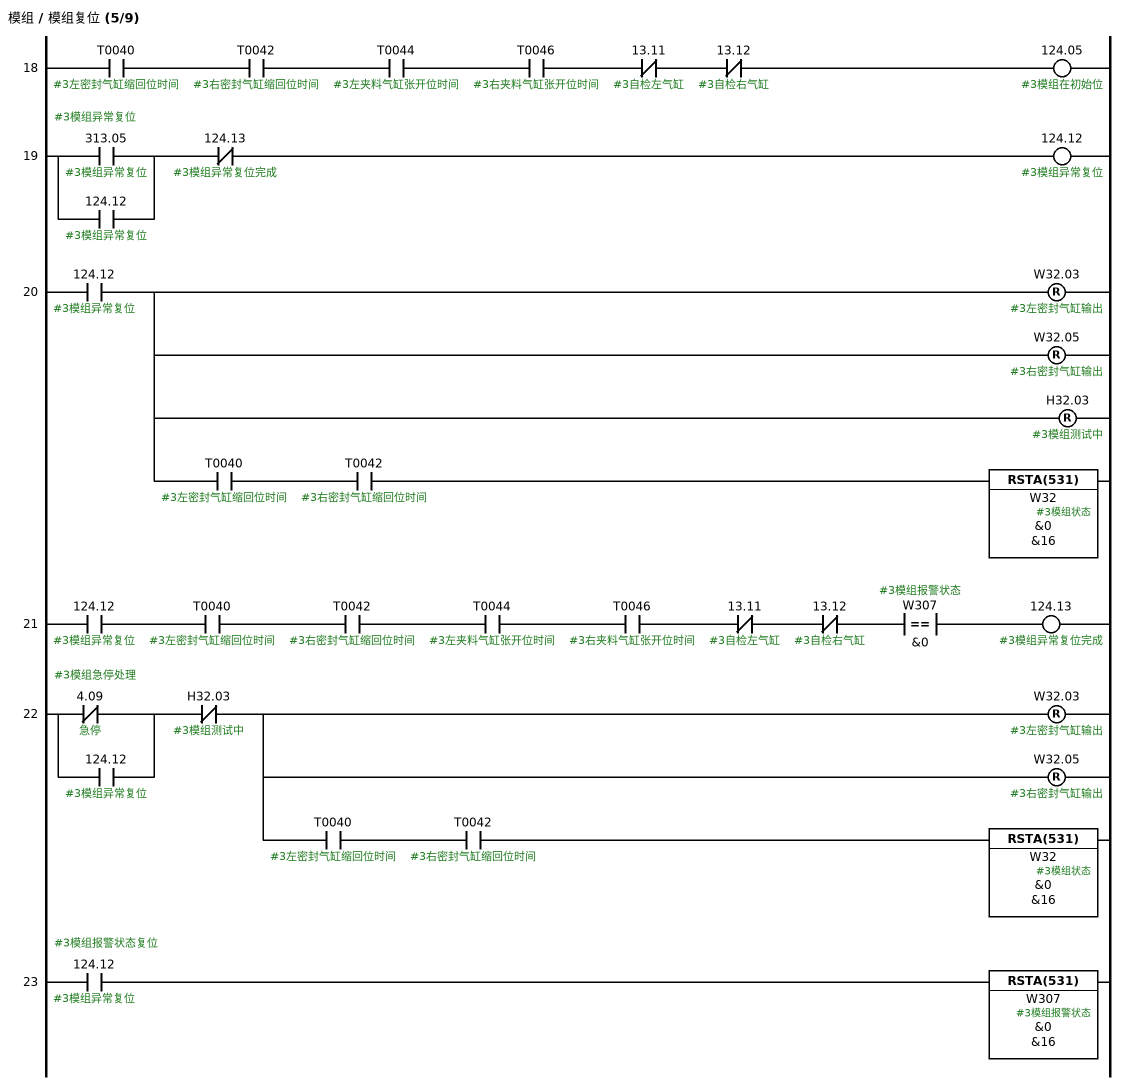
; rung 18
LD T0040  ; #3左密封气缸缩回位时间
AND T0042  ; #3右密封气缸缩回位时间
AND T0044  ; #3左夹料气缸张开位时间
AND T0046  ; #3右夹料气缸张开位时间
ANDNOT 13.11  ; #3自检左气缸
ANDNOT 13.12  ; #3自检右气缸
OUT 124.05  ; #3模组在初始位
; rung 19: #3模组异常复位
LD 313.05  ; #3模组异常复位
OR 124.12  ; #3模组异常复位
ANDNOT 124.13  ; #3模组异常复位完成
OUT 124.12  ; #3模组异常复位
; rung 20
LD 124.12  ; #3模组异常复位
RSET W32.03  ; #3左密封气缸输出
RSET W32.05  ; #3右密封气缸输出
RSET H32.03  ; #3模组测试中
AND T0040  ; #3左密封气缸缩回位时间
AND T0042  ; #3右密封气缸缩回位时间
RSTA(531) W32 &0 &16  ; #3模组状态
; rung 21
LD 124.12  ; #3模组异常复位
AND T0040  ; #3左密封气缸缩回位时间
AND T0042  ; #3右密封气缸缩回位时间
AND T0044  ; #3左夹料气缸张开位时间
AND T0046  ; #3右夹料气缸张开位时间
ANDNOT 13.11  ; #3自检左气缸
ANDNOT 13.12  ; #3自检右气缸
AND=(300) W307 &0  ; #3模组报警状态
OUT 124.13  ; #3模组异常复位完成
; rung 22: #3模组急停处理
LDNOT 4.09  ; 急停
OR 124.12  ; #3模组异常复位
ANDNOT H32.03  ; #3模组测试中
RSET W32.03  ; #3左密封气缸输出
RSET W32.05  ; #3右密封气缸输出
AND T0040  ; #3左密封气缸缩回位时间
AND T0042  ; #3右密封气缸缩回位时间
RSTA(531) W32 &0 &16  ; #3模组状态
; rung 23: #3模组报警状态复位
LD 124.12  ; #3模组异常复位
RSTA(531) W307 &0 &16  ; #3模组报警状态

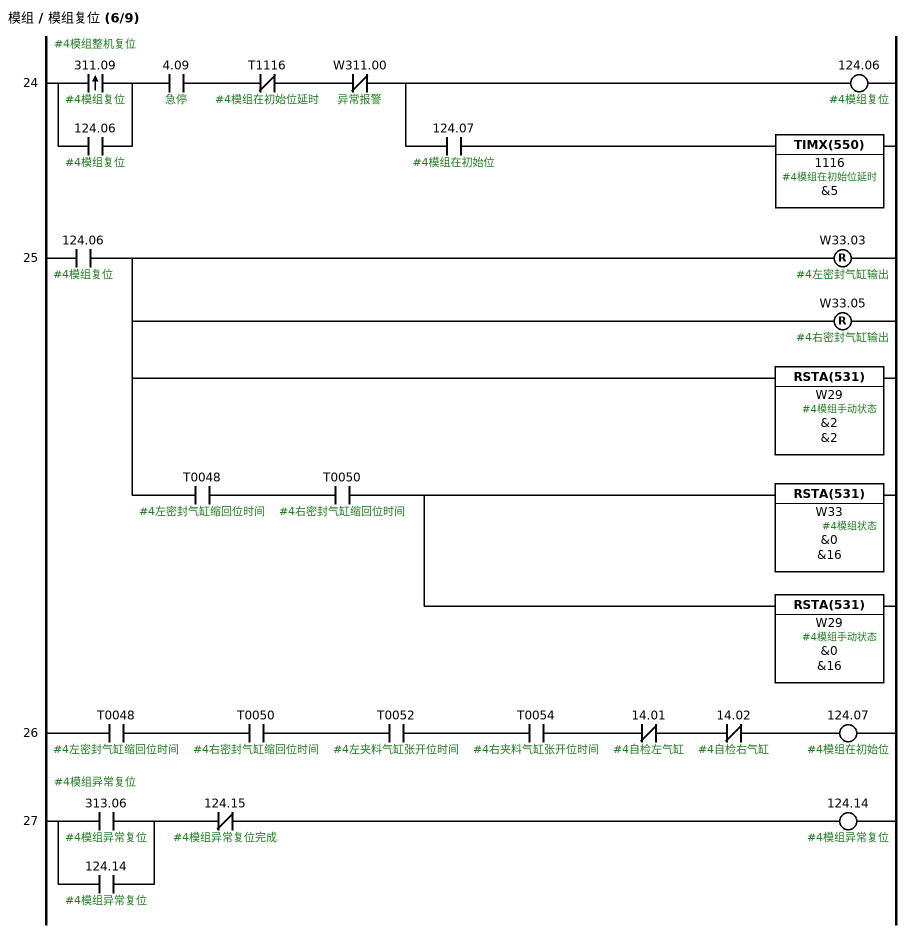
; rung 24: #4模组整机复位
@LD 311.09  ; #4模组复位
OR 124.06  ; #4模组复位
AND 4.09  ; 急停
ANDNOT T1116  ; #4模组在初始位延时
ANDNOT W311.00  ; 异常报警
OUT 124.06  ; #4模组复位
AND 124.07  ; #4模组在初始位
TIMX(550) 1116 &5  ; #4模组在初始位延时
; rung 25
LD 124.06  ; #4模组复位
RSET W33.03  ; #4左密封气缸输出
RSET W33.05  ; #4右密封气缸输出
RSTA(531) W29 &2 &2  ; #4模组手动状态
AND T0048  ; #4左密封气缸缩回位时间
AND T0050  ; #4右密封气缸缩回位时间
RSTA(531) W33 &0 &16  ; #4模组状态
RSTA(531) W29 &0 &16  ; #4模组手动状态
; rung 26
LD T0048  ; #4左密封气缸缩回位时间
AND T0050  ; #4右密封气缸缩回位时间
AND T0052  ; #4左夹料气缸张开位时间
AND T0054  ; #4右夹料气缸张开位时间
ANDNOT 14.01  ; #4自检左气缸
ANDNOT 14.02  ; #4自检右气缸
OUT 124.07  ; #4模组在初始位
; rung 27: #4模组异常复位
LD 313.06  ; #4模组异常复位
OR 124.14  ; #4模组异常复位
ANDNOT 124.15  ; #4模组异常复位完成
OUT 124.14  ; #4模组异常复位

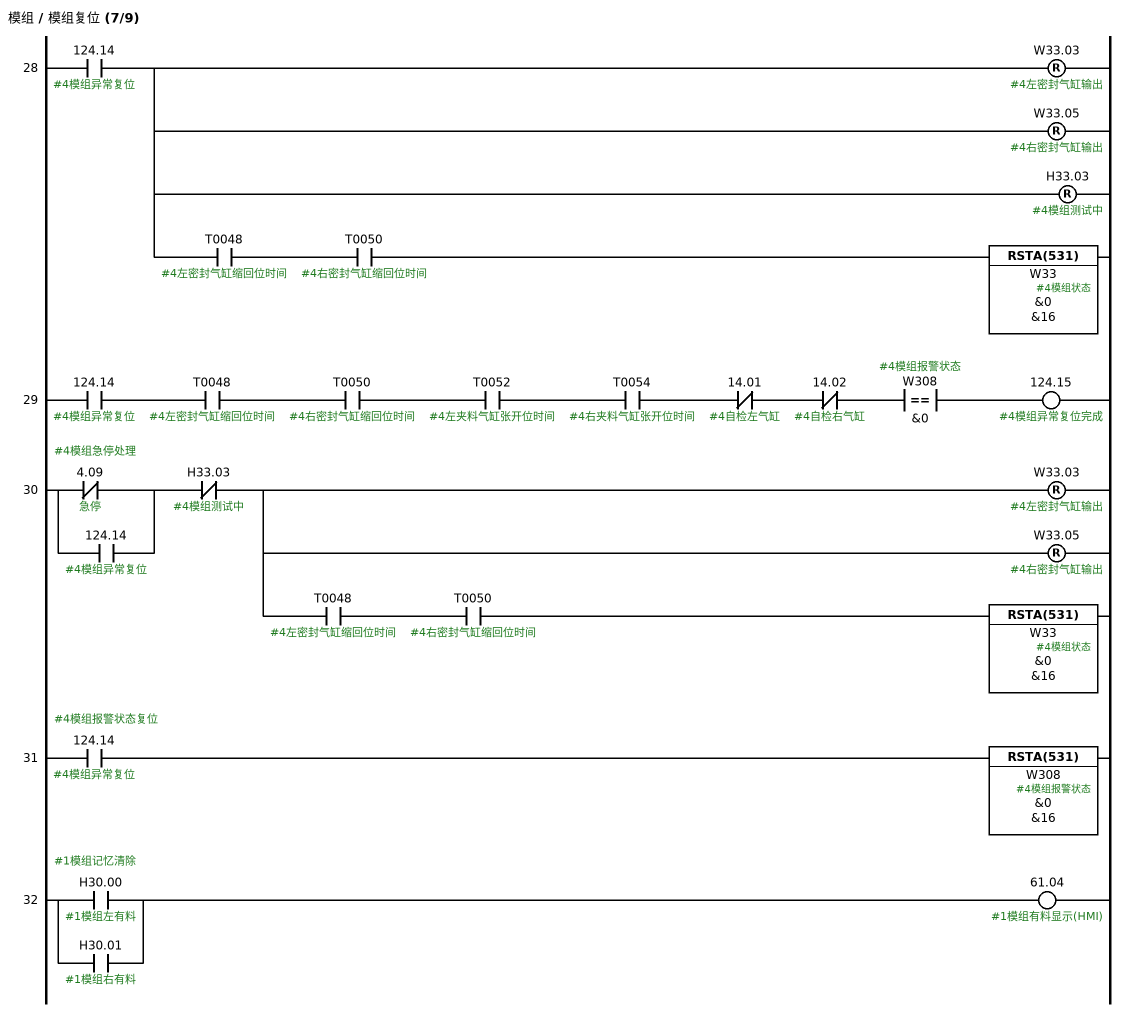
; rung 28
LD 124.14  ; #4模组异常复位
RSET W33.03  ; #4左密封气缸输出
RSET W33.05  ; #4右密封气缸输出
RSET H33.03  ; #4模组测试中
AND T0048  ; #4左密封气缸缩回位时间
AND T0050  ; #4右密封气缸缩回位时间
RSTA(531) W33 &0 &16  ; #4模组状态
; rung 29
LD 124.14  ; #4模组异常复位
AND T0048  ; #4左密封气缸缩回位时间
AND T0050  ; #4右密封气缸缩回位时间
AND T0052  ; #4左夹料气缸张开位时间
AND T0054  ; #4右夹料气缸张开位时间
ANDNOT 14.01  ; #4自检左气缸
ANDNOT 14.02  ; #4自检右气缸
AND=(300) W308 &0  ; #4模组报警状态
OUT 124.15  ; #4模组异常复位完成
; rung 30: #4模组急停处理
LDNOT 4.09  ; 急停
OR 124.14  ; #4模组异常复位
ANDNOT H33.03  ; #4模组测试中
RSET W33.03  ; #4左密封气缸输出
RSET W33.05  ; #4右密封气缸输出
AND T0048  ; #4左密封气缸缩回位时间
AND T0050  ; #4右密封气缸缩回位时间
RSTA(531) W33 &0 &16  ; #4模组状态
; rung 31: #4模组报警状态复位
LD 124.14  ; #4模组异常复位
RSTA(531) W308 &0 &16  ; #4模组报警状态
; rung 32: #1模组记忆清除
LD H30.00  ; #1模组左有料
OR H30.01  ; #1模组右有料
OUT 61.04  ; #1模组有料显示(HMI)

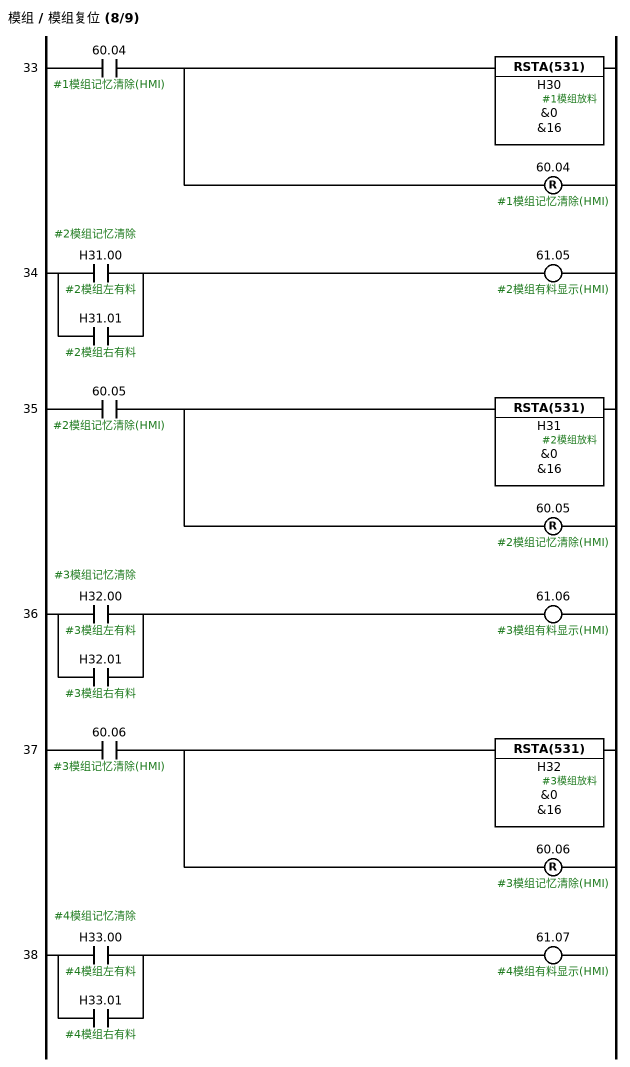
; rung 33
LD 60.04  ; #1模组记忆清除(HMI)
RSTA(531) H30 &0 &16  ; #1模组放料
RSET 60.04  ; #1模组记忆清除(HMI)
; rung 34: #2模组记忆清除
LD H31.00  ; #2模组左有料
OR H31.01  ; #2模组右有料
OUT 61.05  ; #2模组有料显示(HMI)
; rung 35
LD 60.05  ; #2模组记忆清除(HMI)
RSTA(531) H31 &0 &16  ; #2模组放料
RSET 60.05  ; #2模组记忆清除(HMI)
; rung 36: #3模组记忆清除
LD H32.00  ; #3模组左有料
OR H32.01  ; #3模组右有料
OUT 61.06  ; #3模组有料显示(HMI)
; rung 37
LD 60.06  ; #3模组记忆清除(HMI)
RSTA(531) H32 &0 &16  ; #3模组放料
RSET 60.06  ; #3模组记忆清除(HMI)
; rung 38: #4模组记忆清除
LD H33.00  ; #4模组左有料
OR H33.01  ; #4模组右有料
OUT 61.07  ; #4模组有料显示(HMI)

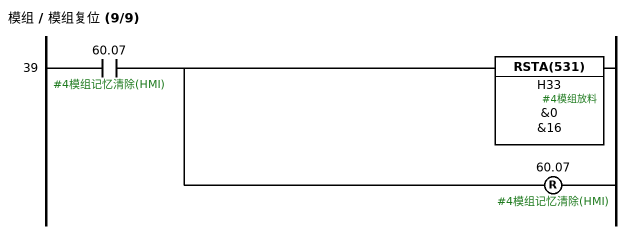
; rung 39
LD 60.07  ; #4模组记忆清除(HMI)
RSTA(531) H33 &0 &16  ; #4模组放料
RSET 60.07  ; #4模组记忆清除(HMI)

### Section END
; rung 0
END(001)

## Program 龙门机械手 (cyclic task 7)
Local symbols
P_on BOOL

### Section 龙门、料盒升降手动

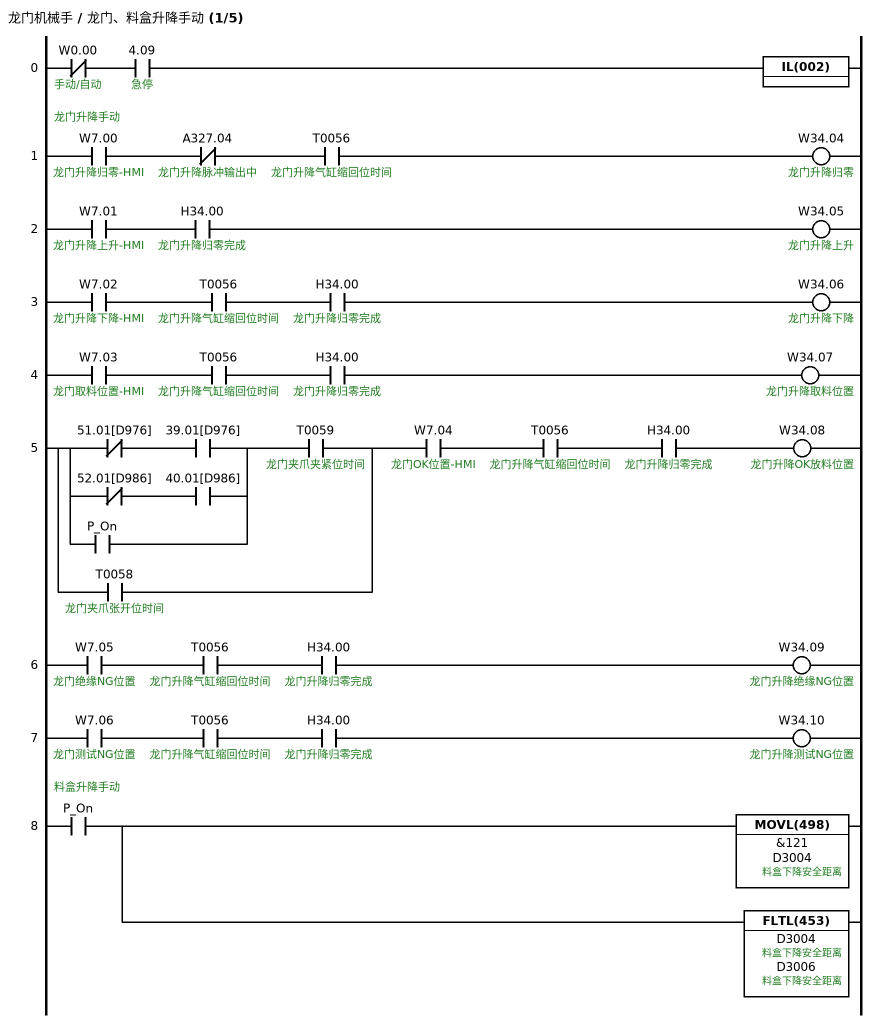
; rung 0
LDNOT W0.00  ; 手动/自动
AND 4.09  ; 急停
IL(002)
; rung 1: 龙门升降手动
LD W7.00  ; 龙门升降归零-HMI
ANDNOT A327.04  ; 龙门升降脉冲输出中
AND T0056  ; 龙门升降气缸缩回位时间
OUT W34.04  ; 龙门升降归零
; rung 2
LD W7.01  ; 龙门升降上升-HMI
AND H34.00  ; 龙门升降归零完成
OUT W34.05  ; 龙门升降上升
; rung 3
LD W7.02  ; 龙门升降下降-HMI
AND T0056  ; 龙门升降气缸缩回位时间
AND H34.00  ; 龙门升降归零完成
OUT W34.06  ; 龙门升降下降
; rung 4
LD W7.03  ; 龙门取料位置-HMI
AND T0056  ; 龙门升降气缸缩回位时间
AND H34.00  ; 龙门升降归零完成
OUT W34.07  ; 龙门升降取料位置
; rung 5
LDNOT 51.01[D976]
AND 39.01[D976]
LDNOT 52.01[D986]
AND 40.01[D986]
ORLD
OR P_On
AND T0059  ; 龙门夹爪夹紧位时间
OR T0058  ; 龙门夹爪张开位时间
AND W7.04  ; 龙门OK位置-HMI
AND T0056  ; 龙门升降气缸缩回位时间
AND H34.00  ; 龙门升降归零完成
OUT W34.08  ; 龙门升降OK放料位置
; rung 6
LD W7.05  ; 龙门绝缘NG位置
AND T0056  ; 龙门升降气缸缩回位时间
AND H34.00  ; 龙门升降归零完成
OUT W34.09  ; 龙门升降绝缘NG位置
; rung 7
LD W7.06  ; 龙门测试NG位置
AND T0056  ; 龙门升降气缸缩回位时间
AND H34.00  ; 龙门升降归零完成
OUT W34.10  ; 龙门升降测试NG位置
; rung 8: 料盒升降手动
LD P_On
MOVL(498) &121 D3004  ; 料盒下降安全距离
FLTL(453) D3004 D3006  ; 料盒下降安全距离

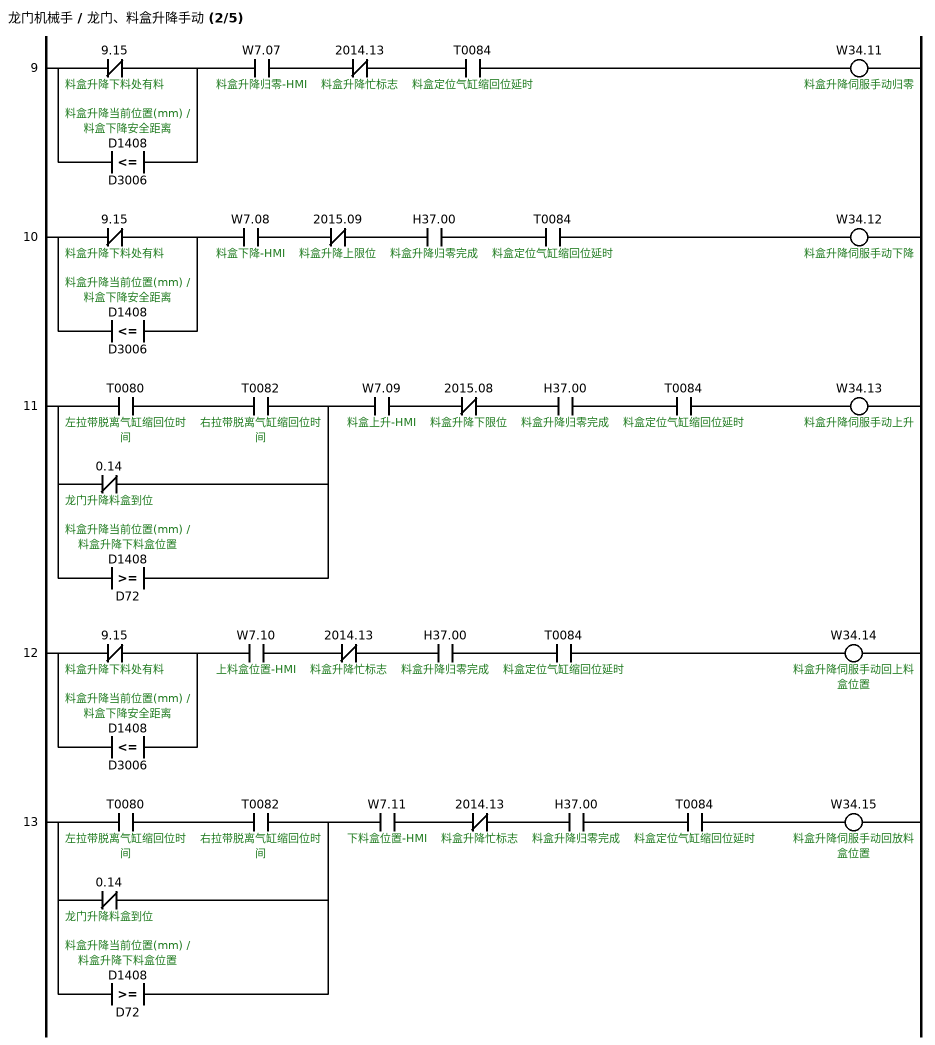
; rung 9
LDNOT 9.15  ; 料盒升降下料处有料
OR<=F(332) D1408 D3006  ; 料盒升降当前位置(mm), 料盒下降安全距离
AND W7.07  ; 料盒升降归零-HMI
ANDNOT 2014.13  ; 料盒升降忙标志
AND T0084  ; 料盒定位气缸缩回位延时
OUT W34.11  ; 料盒升降伺服手动归零
; rung 10
LDNOT 9.15  ; 料盒升降下料处有料
OR<=F(332) D1408 D3006  ; 料盒升降当前位置(mm), 料盒下降安全距离
AND W7.08  ; 料盒下降-HMI
ANDNOT 2015.09  ; 料盒升降上限位
AND H37.00  ; 料盒升降归零完成
AND T0084  ; 料盒定位气缸缩回位延时
OUT W34.12  ; 料盒升降伺服手动下降
; rung 11
LD T0080  ; 左拉带脱离气缸缩回位时间
AND T0082  ; 右拉带脱离气缸缩回位时间
ORNOT 0.14  ; 龙门升降料盒到位
OR>=F(334) D1408 D72  ; 料盒升降当前位置(mm), 料盒升降下料盒位置
AND W7.09  ; 料盒上升-HMI
ANDNOT 2015.08  ; 料盒升降下限位
AND H37.00  ; 料盒升降归零完成
AND T0084  ; 料盒定位气缸缩回位延时
OUT W34.13  ; 料盒升降伺服手动上升
; rung 12
LDNOT 9.15  ; 料盒升降下料处有料
OR<=F(332) D1408 D3006  ; 料盒升降当前位置(mm), 料盒下降安全距离
AND W7.10  ; 上料盒位置-HMI
ANDNOT 2014.13  ; 料盒升降忙标志
AND H37.00  ; 料盒升降归零完成
AND T0084  ; 料盒定位气缸缩回位延时
OUT W34.14  ; 料盒升降伺服手动回上料盒位置
; rung 13
LD T0080  ; 左拉带脱离气缸缩回位时间
AND T0082  ; 右拉带脱离气缸缩回位时间
ORNOT 0.14  ; 龙门升降料盒到位
OR>=F(334) D1408 D72  ; 料盒升降当前位置(mm), 料盒升降下料盒位置
AND W7.11  ; 下料盒位置-HMI
ANDNOT 2014.13  ; 料盒升降忙标志
AND H37.00  ; 料盒升降归零完成
AND T0084  ; 料盒定位气缸缩回位延时
OUT W34.15  ; 料盒升降伺服手动回放料盒位置

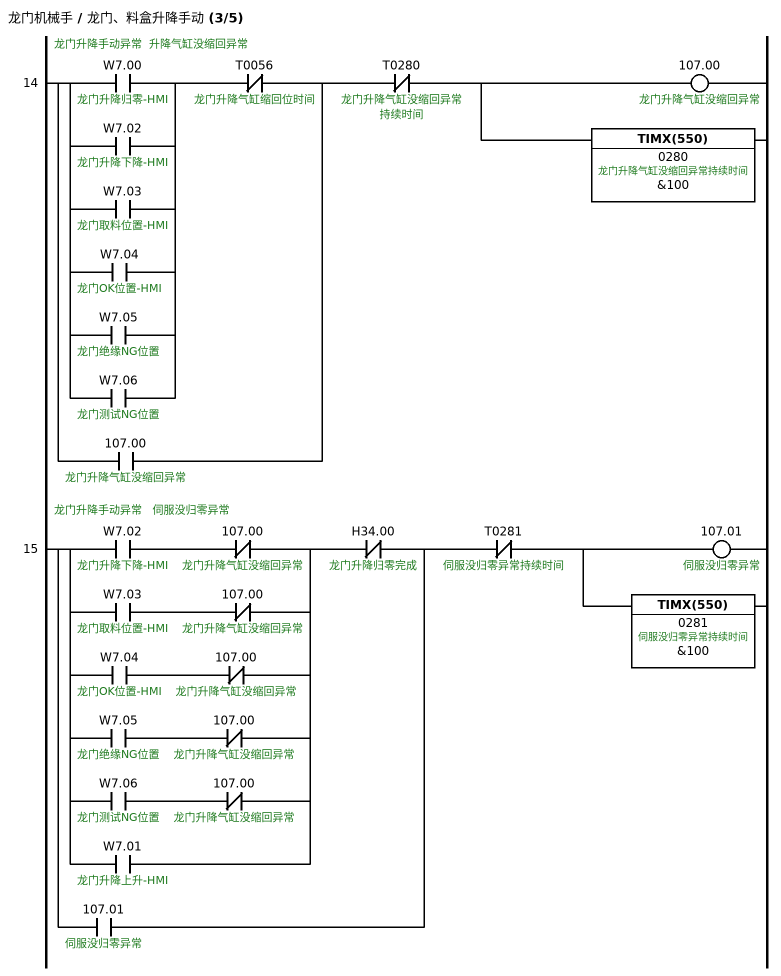
; rung 14: 龙门升降手动异常  升降气缸没缩回异常
LD W7.00  ; 龙门升降归零-HMI
OR W7.02  ; 龙门升降下降-HMI
OR W7.03  ; 龙门取料位置-HMI
OR W7.04  ; 龙门OK位置-HMI
OR W7.05  ; 龙门绝缘NG位置
OR W7.06  ; 龙门测试NG位置
ANDNOT T0056  ; 龙门升降气缸缩回位时间
OR 107.00  ; 龙门升降气缸没缩回异常
ANDNOT T0280  ; 龙门升降气缸没缩回异常持续时间
OUT 107.00  ; 龙门升降气缸没缩回异常
TIMX(550) 0280 &100  ; 龙门升降气缸没缩回异常持续时间
; rung 15: 龙门升降手动异常   伺服没归零异常
LD W7.02  ; 龙门升降下降-HMI
ANDNOT 107.00  ; 龙门升降气缸没缩回异常
LD W7.03  ; 龙门取料位置-HMI
ANDNOT 107.00  ; 龙门升降气缸没缩回异常
ORLD
LD W7.04  ; 龙门OK位置-HMI
ANDNOT 107.00  ; 龙门升降气缸没缩回异常
ORLD
LD W7.05  ; 龙门绝缘NG位置
ANDNOT 107.00  ; 龙门升降气缸没缩回异常
ORLD
LD W7.06  ; 龙门测试NG位置
ANDNOT 107.00  ; 龙门升降气缸没缩回异常
ORLD
OR W7.01  ; 龙门升降上升-HMI
ANDNOT H34.00  ; 龙门升降归零完成
OR 107.01  ; 伺服没归零异常
ANDNOT T0281  ; 伺服没归零异常持续时间
OUT 107.01  ; 伺服没归零异常
TIMX(550) 0281 &100  ; 伺服没归零异常持续时间

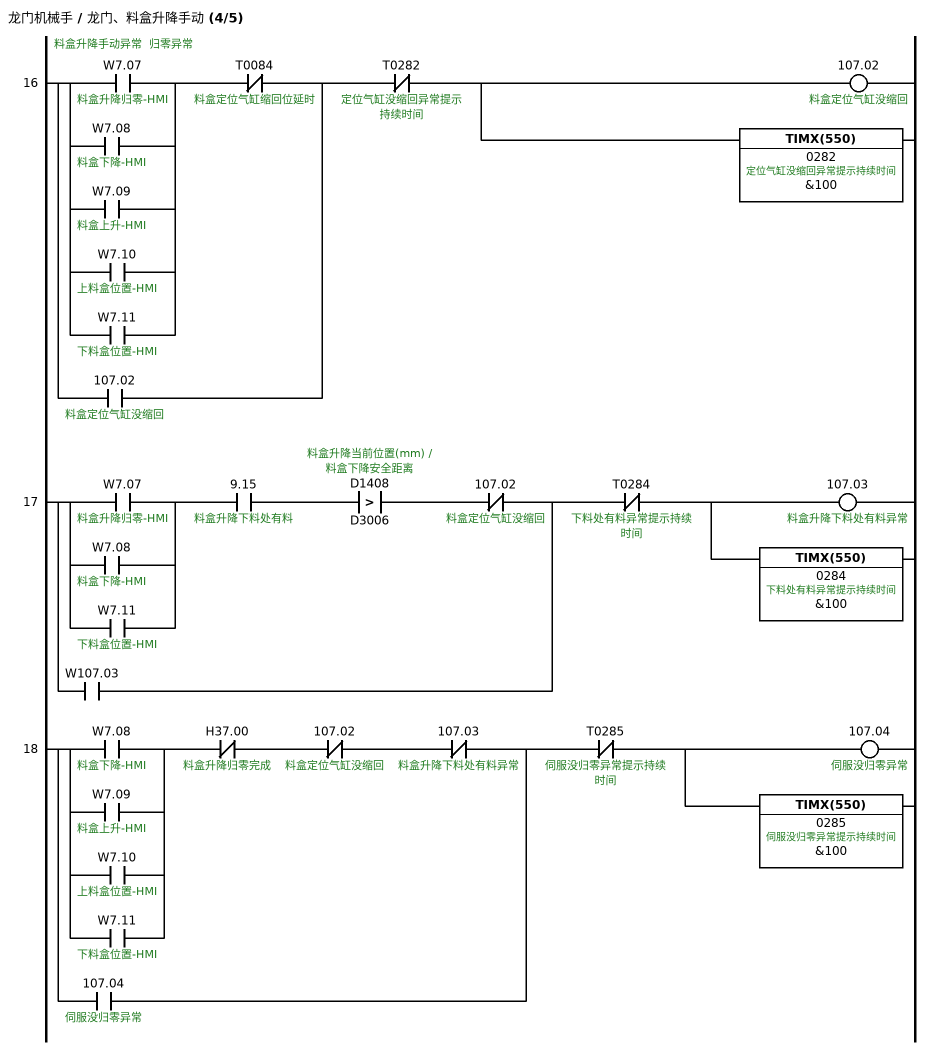
; rung 16: 料盒升降手动异常  归零异常
LD W7.07  ; 料盒升降归零-HMI
OR W7.08  ; 料盒下降-HMI
OR W7.09  ; 料盒上升-HMI
OR W7.10  ; 上料盒位置-HMI
OR W7.11  ; 下料盒位置-HMI
ANDNOT T0084  ; 料盒定位气缸缩回位延时
OR 107.02  ; 料盒定位气缸没缩回
ANDNOT T0282  ; 定位气缸没缩回异常提示持续时间
OUT 107.02  ; 料盒定位气缸没缩回
TIMX(550) 0282 &100  ; 定位气缸没缩回异常提示持续时间
; rung 17
LD W7.07  ; 料盒升降归零-HMI
OR W7.08  ; 料盒下降-HMI
OR W7.11  ; 下料盒位置-HMI
AND 9.15  ; 料盒升降下料处有料
AND>F(333) D1408 D3006  ; 料盒升降当前位置(mm), 料盒下降安全距离
ANDNOT 107.02  ; 料盒定位气缸没缩回
OR W107.03
ANDNOT T0284  ; 下料处有料异常提示持续时间
OUT 107.03  ; 料盒升降下料处有料异常
TIMX(550) 0284 &100  ; 下料处有料异常提示持续时间
; rung 18
LD W7.08  ; 料盒下降-HMI
OR W7.09  ; 料盒上升-HMI
OR W7.10  ; 上料盒位置-HMI
OR W7.11  ; 下料盒位置-HMI
ANDNOT H37.00  ; 料盒升降归零完成
ANDNOT 107.02  ; 料盒定位气缸没缩回
ANDNOT 107.03  ; 料盒升降下料处有料异常
OR 107.04  ; 伺服没归零异常
ANDNOT T0285  ; 伺服没归零异常提示持续时间
OUT 107.04  ; 伺服没归零异常
TIMX(550) 0285 &100  ; 伺服没归零异常提示持续时间

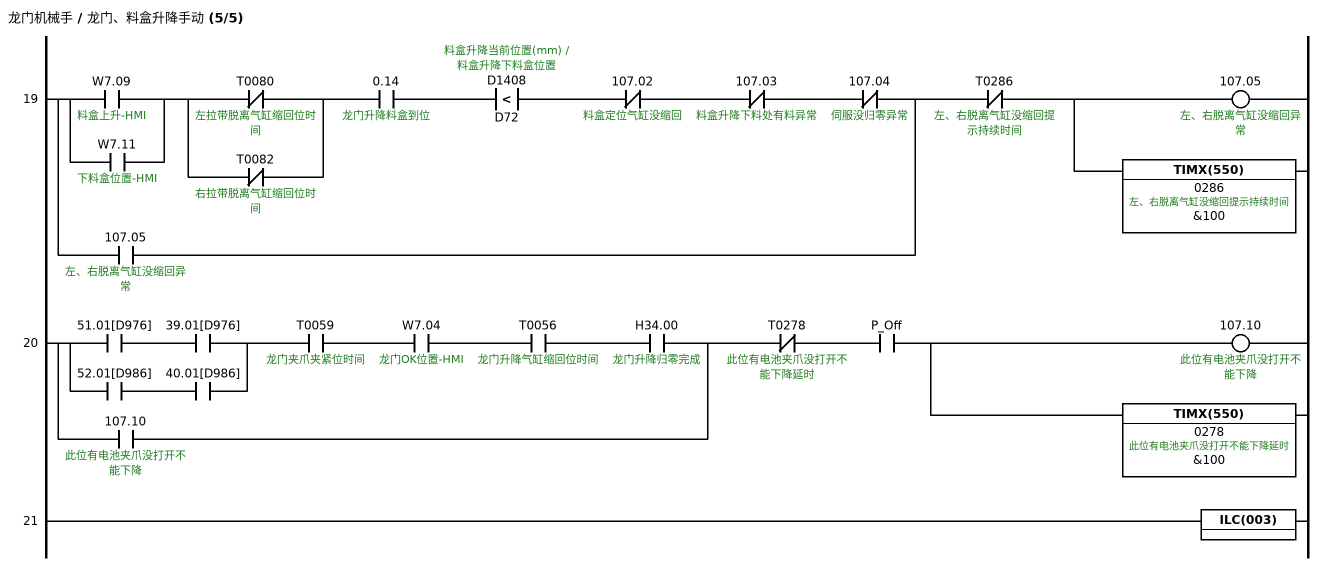
; rung 19
LD W7.09  ; 料盒上升-HMI
OR W7.11  ; 下料盒位置-HMI
LDNOT T0080  ; 左拉带脱离气缸缩回位时间
ORNOT T0082  ; 右拉带脱离气缸缩回位时间
ANDLD
AND 0.14  ; 龙门升降料盒到位
AND<F(331) D1408 D72  ; 料盒升降当前位置(mm), 料盒升降下料盒位置
ANDNOT 107.02  ; 料盒定位气缸没缩回
ANDNOT 107.03  ; 料盒升降下料处有料异常
ANDNOT 107.04  ; 伺服没归零异常
OR 107.05  ; 左、右脱离气缸没缩回异常
ANDNOT T0286  ; 左、右脱离气缸没缩回提示持续时间
OUT 107.05  ; 左、右脱离气缸没缩回异常
TIMX(550) 0286 &100  ; 左、右脱离气缸没缩回提示持续时间
; rung 20
LD 51.01[D976]
AND 39.01[D976]
LD 52.01[D986]
AND 40.01[D986]
ORLD
AND T0059  ; 龙门夹爪夹紧位时间
AND W7.04  ; 龙门OK位置-HMI
AND T0056  ; 龙门升降气缸缩回位时间
AND H34.00  ; 龙门升降归零完成
OR 107.10  ; 此位有电池夹爪没打开不能下降
ANDNOT T0278  ; 此位有电池夹爪没打开不能下降延时
AND P_Off
OUT 107.10  ; 此位有电池夹爪没打开不能下降
TIMX(550) 0278 &100  ; 此位有电池夹爪没打开不能下降延时
; rung 21
ILC(003)

### Section 龙门前后、左右手动

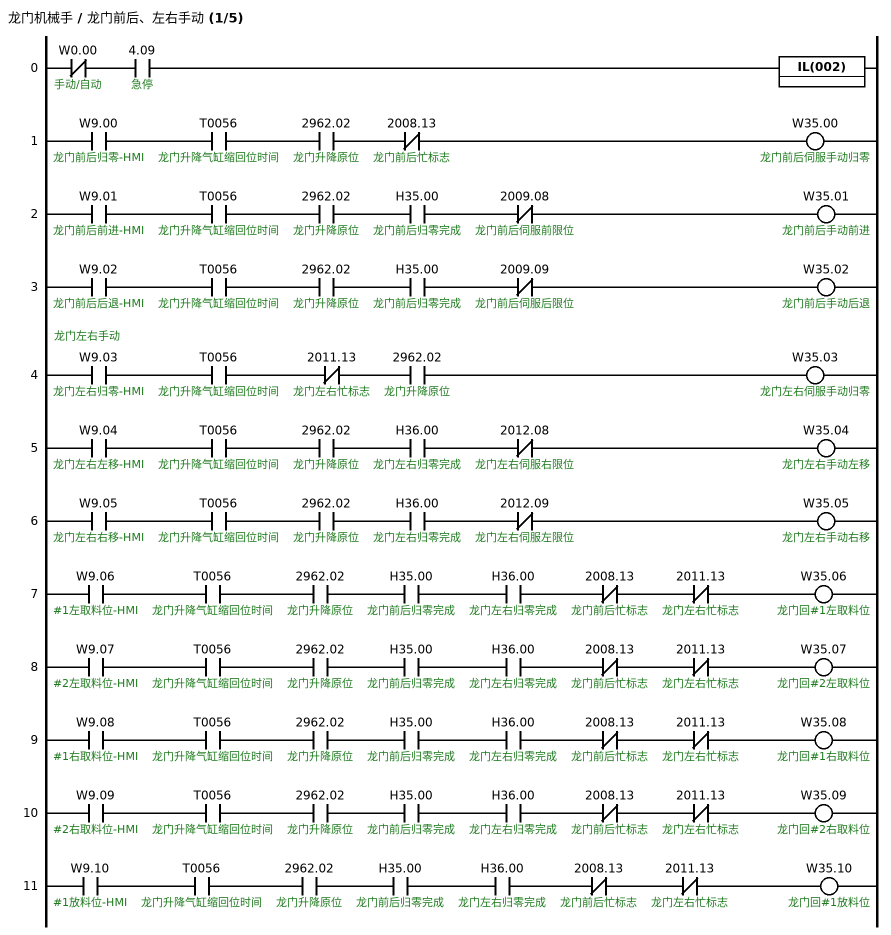
; rung 0
LDNOT W0.00  ; 手动/自动
AND 4.09  ; 急停
IL(002)
; rung 1
LD W9.00  ; 龙门前后归零-HMI
AND T0056  ; 龙门升降气缸缩回位时间
AND 2962.02  ; 龙门升降原位
ANDNOT 2008.13  ; 龙门前后忙标志
OUT W35.00  ; 龙门前后伺服手动归零
; rung 2
LD W9.01  ; 龙门前后前进-HMI
AND T0056  ; 龙门升降气缸缩回位时间
AND 2962.02  ; 龙门升降原位
AND H35.00  ; 龙门前后归零完成
ANDNOT 2009.08  ; 龙门前后伺服前限位
OUT W35.01  ; 龙门前后手动前进
; rung 3
LD W9.02  ; 龙门前后后退-HMI
AND T0056  ; 龙门升降气缸缩回位时间
AND 2962.02  ; 龙门升降原位
AND H35.00  ; 龙门前后归零完成
ANDNOT 2009.09  ; 龙门前后伺服后限位
OUT W35.02  ; 龙门前后手动后退
; rung 4: 龙门左右手动
LD W9.03  ; 龙门左右归零-HMI
AND T0056  ; 龙门升降气缸缩回位时间
ANDNOT 2011.13  ; 龙门左右忙标志
AND 2962.02  ; 龙门升降原位
OUT W35.03  ; 龙门左右伺服手动归零
; rung 5
LD W9.04  ; 龙门左右左移-HMI
AND T0056  ; 龙门升降气缸缩回位时间
AND 2962.02  ; 龙门升降原位
AND H36.00  ; 龙门左右归零完成
ANDNOT 2012.08  ; 龙门左右伺服右限位
OUT W35.04  ; 龙门左右手动左移
; rung 6
LD W9.05  ; 龙门左右右移-HMI
AND T0056  ; 龙门升降气缸缩回位时间
AND 2962.02  ; 龙门升降原位
AND H36.00  ; 龙门左右归零完成
ANDNOT 2012.09  ; 龙门左右伺服左限位
OUT W35.05  ; 龙门左右手动右移
; rung 7
LD W9.06  ; #1左取料位-HMI
AND T0056  ; 龙门升降气缸缩回位时间
AND 2962.02  ; 龙门升降原位
AND H35.00  ; 龙门前后归零完成
AND H36.00  ; 龙门左右归零完成
ANDNOT 2008.13  ; 龙门前后忙标志
ANDNOT 2011.13  ; 龙门左右忙标志
OUT W35.06  ; 龙门回#1左取料位
; rung 8
LD W9.07  ; #2左取料位-HMI
AND T0056  ; 龙门升降气缸缩回位时间
AND 2962.02  ; 龙门升降原位
AND H35.00  ; 龙门前后归零完成
AND H36.00  ; 龙门左右归零完成
ANDNOT 2008.13  ; 龙门前后忙标志
ANDNOT 2011.13  ; 龙门左右忙标志
OUT W35.07  ; 龙门回#2左取料位
; rung 9
LD W9.08  ; #1右取料位-HMI
AND T0056  ; 龙门升降气缸缩回位时间
AND 2962.02  ; 龙门升降原位
AND H35.00  ; 龙门前后归零完成
AND H36.00  ; 龙门左右归零完成
ANDNOT 2008.13  ; 龙门前后忙标志
ANDNOT 2011.13  ; 龙门左右忙标志
OUT W35.08  ; 龙门回#1右取料位
; rung 10
LD W9.09  ; #2右取料位-HMI
AND T0056  ; 龙门升降气缸缩回位时间
AND 2962.02  ; 龙门升降原位
AND H35.00  ; 龙门前后归零完成
AND H36.00  ; 龙门左右归零完成
ANDNOT 2008.13  ; 龙门前后忙标志
ANDNOT 2011.13  ; 龙门左右忙标志
OUT W35.09  ; 龙门回#2右取料位
; rung 11
LD W9.10  ; #1放料位-HMI
AND T0056  ; 龙门升降气缸缩回位时间
AND 2962.02  ; 龙门升降原位
AND H35.00  ; 龙门前后归零完成
AND H36.00  ; 龙门左右归零完成
ANDNOT 2008.13  ; 龙门前后忙标志
ANDNOT 2011.13  ; 龙门左右忙标志
OUT W35.10  ; 龙门回#1放料位

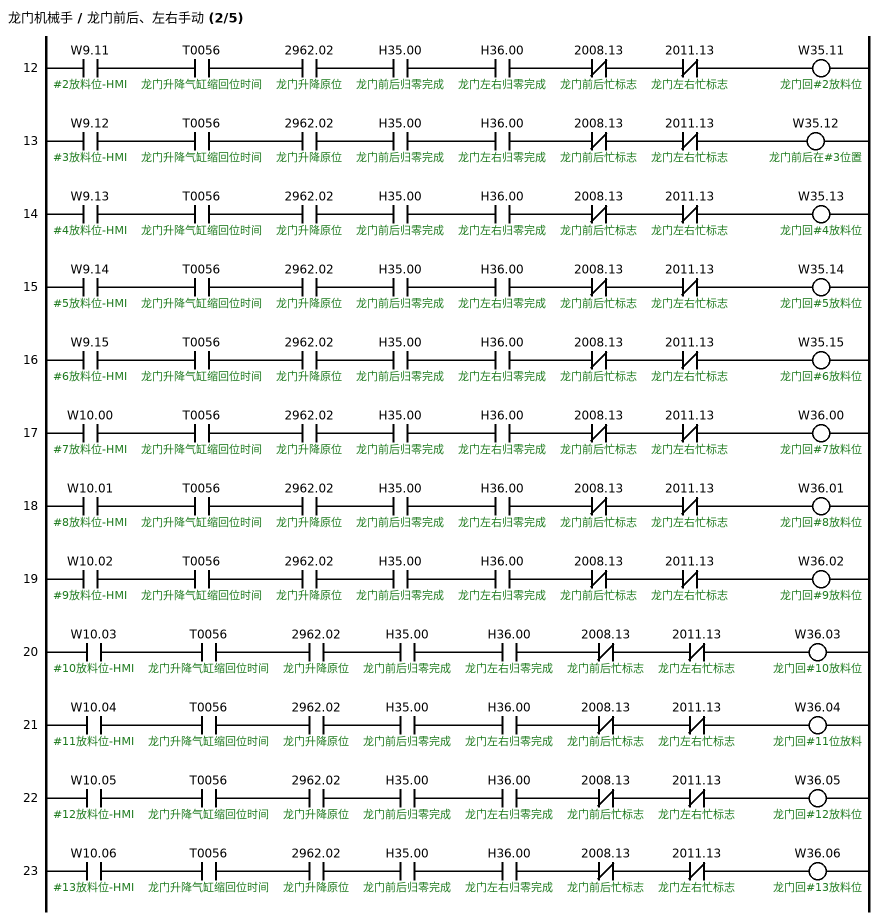
; rung 12
LD W9.11  ; #2放料位-HMI
AND T0056  ; 龙门升降气缸缩回位时间
AND 2962.02  ; 龙门升降原位
AND H35.00  ; 龙门前后归零完成
AND H36.00  ; 龙门左右归零完成
ANDNOT 2008.13  ; 龙门前后忙标志
ANDNOT 2011.13  ; 龙门左右忙标志
OUT W35.11  ; 龙门回#2放料位
; rung 13
LD W9.12  ; #3放料位-HMI
AND T0056  ; 龙门升降气缸缩回位时间
AND 2962.02  ; 龙门升降原位
AND H35.00  ; 龙门前后归零完成
AND H36.00  ; 龙门左右归零完成
ANDNOT 2008.13  ; 龙门前后忙标志
ANDNOT 2011.13  ; 龙门左右忙标志
OUT W35.12  ; 龙门前后在#3位置
; rung 14
LD W9.13  ; #4放料位-HMI
AND T0056  ; 龙门升降气缸缩回位时间
AND 2962.02  ; 龙门升降原位
AND H35.00  ; 龙门前后归零完成
AND H36.00  ; 龙门左右归零完成
ANDNOT 2008.13  ; 龙门前后忙标志
ANDNOT 2011.13  ; 龙门左右忙标志
OUT W35.13  ; 龙门回#4放料位
; rung 15
LD W9.14  ; #5放料位-HMI
AND T0056  ; 龙门升降气缸缩回位时间
AND 2962.02  ; 龙门升降原位
AND H35.00  ; 龙门前后归零完成
AND H36.00  ; 龙门左右归零完成
ANDNOT 2008.13  ; 龙门前后忙标志
ANDNOT 2011.13  ; 龙门左右忙标志
OUT W35.14  ; 龙门回#5放料位
; rung 16
LD W9.15  ; #6放料位-HMI
AND T0056  ; 龙门升降气缸缩回位时间
AND 2962.02  ; 龙门升降原位
AND H35.00  ; 龙门前后归零完成
AND H36.00  ; 龙门左右归零完成
ANDNOT 2008.13  ; 龙门前后忙标志
ANDNOT 2011.13  ; 龙门左右忙标志
OUT W35.15  ; 龙门回#6放料位
; rung 17
LD W10.00  ; #7放料位-HMI
AND T0056  ; 龙门升降气缸缩回位时间
AND 2962.02  ; 龙门升降原位
AND H35.00  ; 龙门前后归零完成
AND H36.00  ; 龙门左右归零完成
ANDNOT 2008.13  ; 龙门前后忙标志
ANDNOT 2011.13  ; 龙门左右忙标志
OUT W36.00  ; 龙门回#7放料位
; rung 18
LD W10.01  ; #8放料位-HMI
AND T0056  ; 龙门升降气缸缩回位时间
AND 2962.02  ; 龙门升降原位
AND H35.00  ; 龙门前后归零完成
AND H36.00  ; 龙门左右归零完成
ANDNOT 2008.13  ; 龙门前后忙标志
ANDNOT 2011.13  ; 龙门左右忙标志
OUT W36.01  ; 龙门回#8放料位
; rung 19
LD W10.02  ; #9放料位-HMI
AND T0056  ; 龙门升降气缸缩回位时间
AND 2962.02  ; 龙门升降原位
AND H35.00  ; 龙门前后归零完成
AND H36.00  ; 龙门左右归零完成
ANDNOT 2008.13  ; 龙门前后忙标志
ANDNOT 2011.13  ; 龙门左右忙标志
OUT W36.02  ; 龙门回#9放料位
; rung 20
LD W10.03  ; #10放料位-HMI
AND T0056  ; 龙门升降气缸缩回位时间
AND 2962.02  ; 龙门升降原位
AND H35.00  ; 龙门前后归零完成
AND H36.00  ; 龙门左右归零完成
ANDNOT 2008.13  ; 龙门前后忙标志
ANDNOT 2011.13  ; 龙门左右忙标志
OUT W36.03  ; 龙门回#10放料位
; rung 21
LD W10.04  ; #11放料位-HMI
AND T0056  ; 龙门升降气缸缩回位时间
AND 2962.02  ; 龙门升降原位
AND H35.00  ; 龙门前后归零完成
AND H36.00  ; 龙门左右归零完成
ANDNOT 2008.13  ; 龙门前后忙标志
ANDNOT 2011.13  ; 龙门左右忙标志
OUT W36.04  ; 龙门回#11位放料
; rung 22
LD W10.05  ; #12放料位-HMI
AND T0056  ; 龙门升降气缸缩回位时间
AND 2962.02  ; 龙门升降原位
AND H35.00  ; 龙门前后归零完成
AND H36.00  ; 龙门左右归零完成
ANDNOT 2008.13  ; 龙门前后忙标志
ANDNOT 2011.13  ; 龙门左右忙标志
OUT W36.05  ; 龙门回#12放料位
; rung 23
LD W10.06  ; #13放料位-HMI
AND T0056  ; 龙门升降气缸缩回位时间
AND 2962.02  ; 龙门升降原位
AND H35.00  ; 龙门前后归零完成
AND H36.00  ; 龙门左右归零完成
ANDNOT 2008.13  ; 龙门前后忙标志
ANDNOT 2011.13  ; 龙门左右忙标志
OUT W36.06  ; 龙门回#13放料位

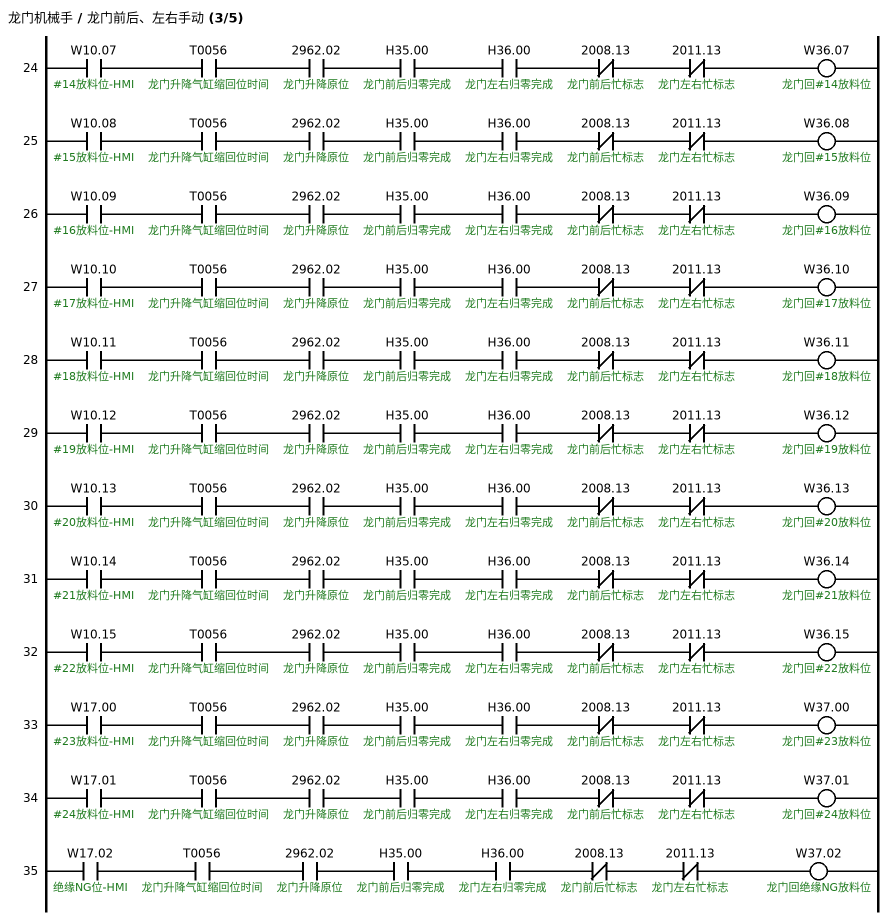
; rung 24
LD W10.07  ; #14放料位-HMI
AND T0056  ; 龙门升降气缸缩回位时间
AND 2962.02  ; 龙门升降原位
AND H35.00  ; 龙门前后归零完成
AND H36.00  ; 龙门左右归零完成
ANDNOT 2008.13  ; 龙门前后忙标志
ANDNOT 2011.13  ; 龙门左右忙标志
OUT W36.07  ; 龙门回#14放料位
; rung 25
LD W10.08  ; #15放料位-HMI
AND T0056  ; 龙门升降气缸缩回位时间
AND 2962.02  ; 龙门升降原位
AND H35.00  ; 龙门前后归零完成
AND H36.00  ; 龙门左右归零完成
ANDNOT 2008.13  ; 龙门前后忙标志
ANDNOT 2011.13  ; 龙门左右忙标志
OUT W36.08  ; 龙门回#15放料位
; rung 26
LD W10.09  ; #16放料位-HMI
AND T0056  ; 龙门升降气缸缩回位时间
AND 2962.02  ; 龙门升降原位
AND H35.00  ; 龙门前后归零完成
AND H36.00  ; 龙门左右归零完成
ANDNOT 2008.13  ; 龙门前后忙标志
ANDNOT 2011.13  ; 龙门左右忙标志
OUT W36.09  ; 龙门回#16放料位
; rung 27
LD W10.10  ; #17放料位-HMI
AND T0056  ; 龙门升降气缸缩回位时间
AND 2962.02  ; 龙门升降原位
AND H35.00  ; 龙门前后归零完成
AND H36.00  ; 龙门左右归零完成
ANDNOT 2008.13  ; 龙门前后忙标志
ANDNOT 2011.13  ; 龙门左右忙标志
OUT W36.10  ; 龙门回#17放料位
; rung 28
LD W10.11  ; #18放料位-HMI
AND T0056  ; 龙门升降气缸缩回位时间
AND 2962.02  ; 龙门升降原位
AND H35.00  ; 龙门前后归零完成
AND H36.00  ; 龙门左右归零完成
ANDNOT 2008.13  ; 龙门前后忙标志
ANDNOT 2011.13  ; 龙门左右忙标志
OUT W36.11  ; 龙门回#18放料位
; rung 29
LD W10.12  ; #19放料位-HMI
AND T0056  ; 龙门升降气缸缩回位时间
AND 2962.02  ; 龙门升降原位
AND H35.00  ; 龙门前后归零完成
AND H36.00  ; 龙门左右归零完成
ANDNOT 2008.13  ; 龙门前后忙标志
ANDNOT 2011.13  ; 龙门左右忙标志
OUT W36.12  ; 龙门回#19放料位
; rung 30
LD W10.13  ; #20放料位-HMI
AND T0056  ; 龙门升降气缸缩回位时间
AND 2962.02  ; 龙门升降原位
AND H35.00  ; 龙门前后归零完成
AND H36.00  ; 龙门左右归零完成
ANDNOT 2008.13  ; 龙门前后忙标志
ANDNOT 2011.13  ; 龙门左右忙标志
OUT W36.13  ; 龙门回#20放料位
; rung 31
LD W10.14  ; #21放料位-HMI
AND T0056  ; 龙门升降气缸缩回位时间
AND 2962.02  ; 龙门升降原位
AND H35.00  ; 龙门前后归零完成
AND H36.00  ; 龙门左右归零完成
ANDNOT 2008.13  ; 龙门前后忙标志
ANDNOT 2011.13  ; 龙门左右忙标志
OUT W36.14  ; 龙门回#21放料位
; rung 32
LD W10.15  ; #22放料位-HMI
AND T0056  ; 龙门升降气缸缩回位时间
AND 2962.02  ; 龙门升降原位
AND H35.00  ; 龙门前后归零完成
AND H36.00  ; 龙门左右归零完成
ANDNOT 2008.13  ; 龙门前后忙标志
ANDNOT 2011.13  ; 龙门左右忙标志
OUT W36.15  ; 龙门回#22放料位
; rung 33
LD W17.00  ; #23放料位-HMI
AND T0056  ; 龙门升降气缸缩回位时间
AND 2962.02  ; 龙门升降原位
AND H35.00  ; 龙门前后归零完成
AND H36.00  ; 龙门左右归零完成
ANDNOT 2008.13  ; 龙门前后忙标志
ANDNOT 2011.13  ; 龙门左右忙标志
OUT W37.00  ; 龙门回#23放料位
; rung 34
LD W17.01  ; #24放料位-HMI
AND T0056  ; 龙门升降气缸缩回位时间
AND 2962.02  ; 龙门升降原位
AND H35.00  ; 龙门前后归零完成
AND H36.00  ; 龙门左右归零完成
ANDNOT 2008.13  ; 龙门前后忙标志
ANDNOT 2011.13  ; 龙门左右忙标志
OUT W37.01  ; 龙门回#24放料位
; rung 35
LD W17.02  ; 绝缘NG位-HMI
AND T0056  ; 龙门升降气缸缩回位时间
AND 2962.02  ; 龙门升降原位
AND H35.00  ; 龙门前后归零完成
AND H36.00  ; 龙门左右归零完成
ANDNOT 2008.13  ; 龙门前后忙标志
ANDNOT 2011.13  ; 龙门左右忙标志
OUT W37.02  ; 龙门回绝缘NG放料位

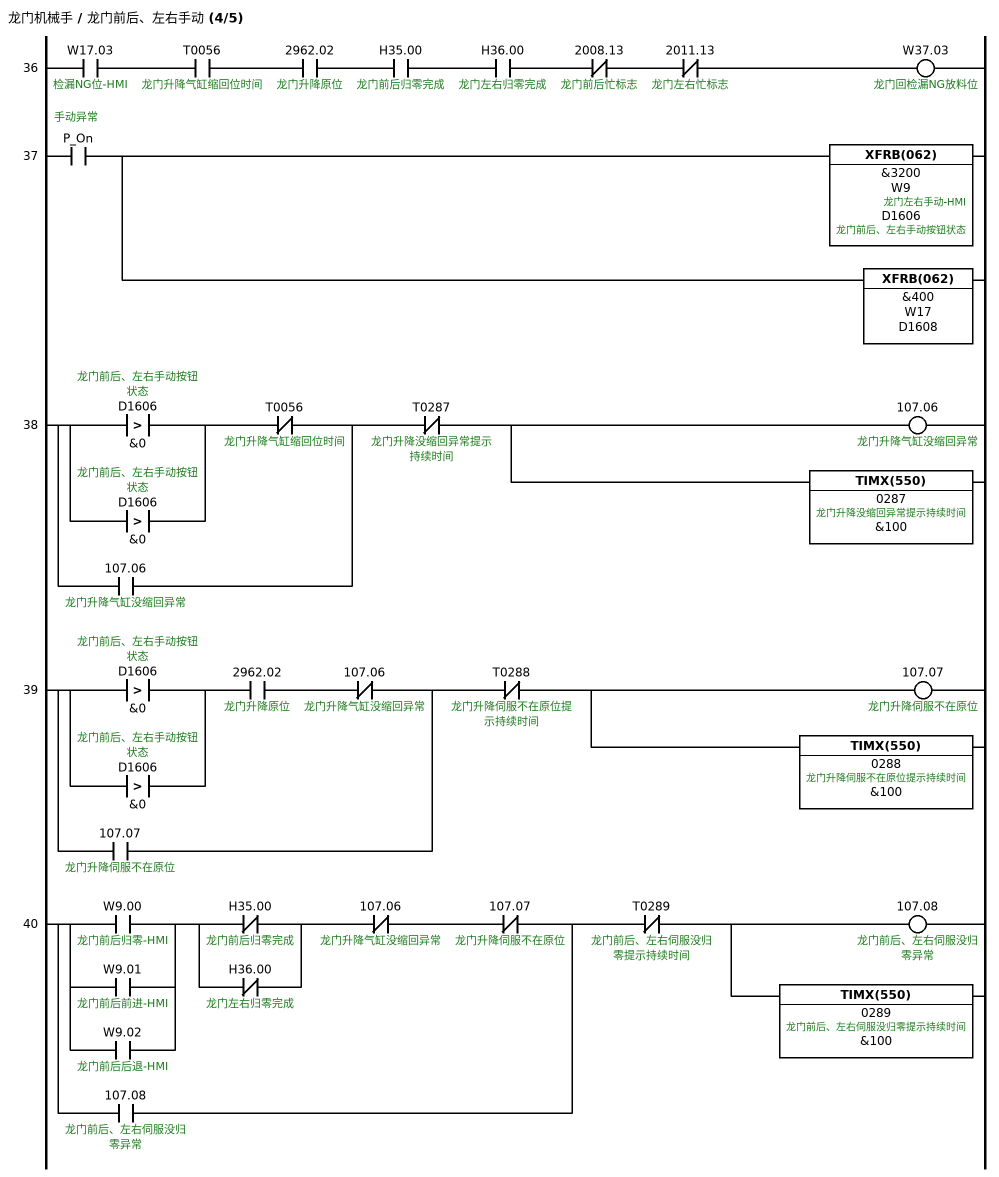
; rung 36
LD W17.03  ; 检漏NG位-HMI
AND T0056  ; 龙门升降气缸缩回位时间
AND 2962.02  ; 龙门升降原位
AND H35.00  ; 龙门前后归零完成
AND H36.00  ; 龙门左右归零完成
ANDNOT 2008.13  ; 龙门前后忙标志
ANDNOT 2011.13  ; 龙门左右忙标志
OUT W37.03  ; 龙门回检漏NG放料位
; rung 37: 手动异常
LD P_On
XFRB(062) &3200 W9 D1606  ; 龙门左右手动-HMI, 龙门前后、左右手动按钮状态
XFRB(062) &400 W17 D1608
; rung 38
LD>(320) D1606 &0  ; 龙门前后、左右手动按钮状态
OR>(320) D1606 &0  ; 龙门前后、左右手动按钮状态
ANDNOT T0056  ; 龙门升降气缸缩回位时间
OR 107.06  ; 龙门升降气缸没缩回异常
ANDNOT T0287  ; 龙门升降没缩回异常提示持续时间
OUT 107.06  ; 龙门升降气缸没缩回异常
TIMX(550) 0287 &100  ; 龙门升降没缩回异常提示持续时间
; rung 39
LD>(320) D1606 &0  ; 龙门前后、左右手动按钮状态
OR>(320) D1606 &0  ; 龙门前后、左右手动按钮状态
AND 2962.02  ; 龙门升降原位
ANDNOT 107.06  ; 龙门升降气缸没缩回异常
OR 107.07  ; 龙门升降伺服不在原位
ANDNOT T0288  ; 龙门升降伺服不在原位提示持续时间
OUT 107.07  ; 龙门升降伺服不在原位
TIMX(550) 0288 &100  ; 龙门升降伺服不在原位提示持续时间
; rung 40
LD W9.00  ; 龙门前后归零-HMI
OR W9.01  ; 龙门前后前进-HMI
OR W9.02  ; 龙门前后后退-HMI
LDNOT H35.00  ; 龙门前后归零完成
ORNOT H36.00  ; 龙门左右归零完成
ANDLD
ANDNOT 107.06  ; 龙门升降气缸没缩回异常
ANDNOT 107.07  ; 龙门升降伺服不在原位
OR 107.08  ; 龙门前后、左右伺服没归零异常
ANDNOT T0289  ; 龙门前后、左右伺服没归零提示持续时间
OUT 107.08  ; 龙门前后、左右伺服没归零异常
TIMX(550) 0289 &100  ; 龙门前后、左右伺服没归零提示持续时间

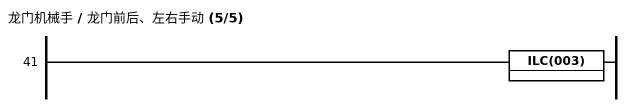
; rung 41
ILC(003)

### Section 龙门升降伺服参数

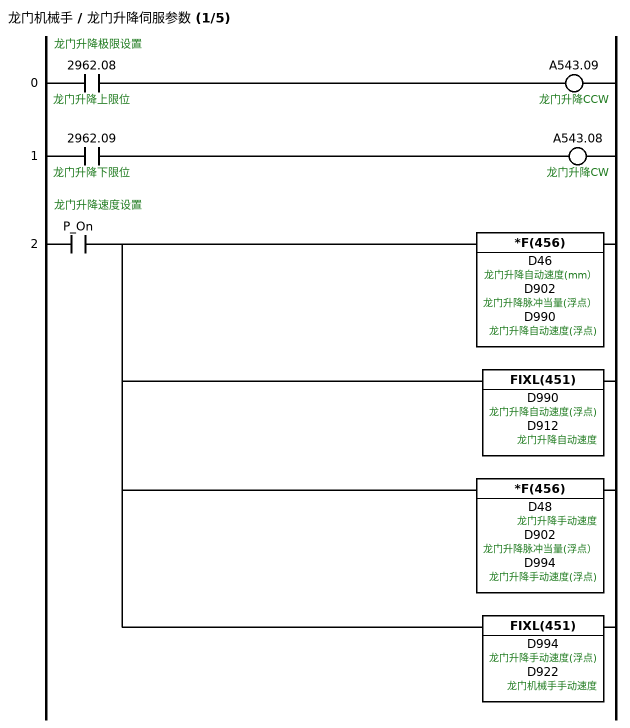
; rung 0: 龙门升降极限设置
LD 2962.08  ; 龙门升降上限位
OUT A543.09  ; 龙门升降CCW
; rung 1
LD 2962.09  ; 龙门升降下限位
OUT A543.08  ; 龙门升降CW
; rung 2: 龙门升降速度设置
LD P_On
*F(456) D46 D902 D990  ; 龙门升降自动速度(mm）, 龙门升降脉冲当量(浮点）, 龙门升降自动速度(浮点)
FIXL(451) D990 D912  ; 龙门升降自动速度(浮点), 龙门升降自动速度
*F(456) D48 D902 D994  ; 龙门升降手动速度, 龙门升降脉冲当量(浮点）, 龙门升降手动速度(浮点)
FIXL(451) D994 D922  ; 龙门升降手动速度(浮点), 龙门机械手手动速度

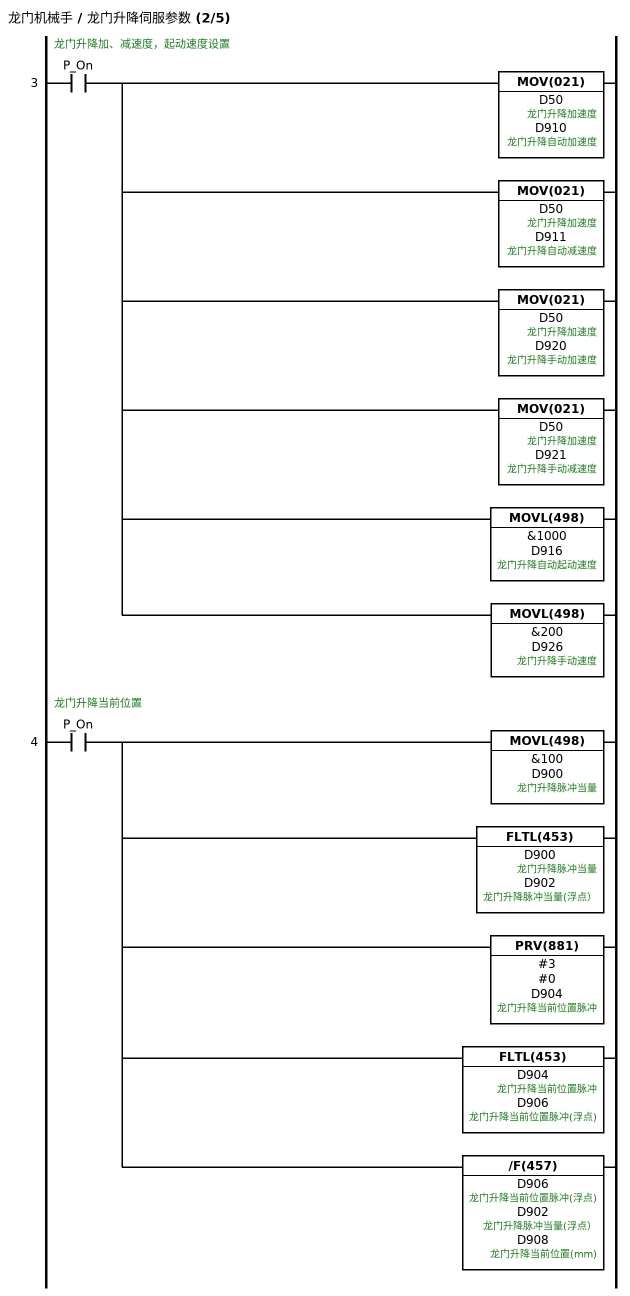
; rung 3: 龙门升降加、减速度，起动速度设置
LD P_On
MOV(021) D50 D910  ; 龙门升降加速度, 龙门升降自动加速度
MOV(021) D50 D911  ; 龙门升降加速度, 龙门升降自动减速度
MOV(021) D50 D920  ; 龙门升降加速度, 龙门升降手动加速度
MOV(021) D50 D921  ; 龙门升降加速度, 龙门升降手动减速度
MOVL(498) &1000 D916  ; 龙门升降自动起动速度
MOVL(498) &200 D926  ; 龙门升降手动速度
; rung 4: 龙门升降当前位置
LD P_On
MOVL(498) &100 D900  ; 龙门升降脉冲当量
FLTL(453) D900 D902  ; 龙门升降脉冲当量, 龙门升降脉冲当量(浮点）
PRV(881) #3 #0 D904  ; 龙门升降当前位置脉冲
FLTL(453) D904 D906  ; 龙门升降当前位置脉冲, 龙门升降当前位置脉冲(浮点)
/F(457) D906 D902 D908  ; 龙门升降当前位置脉冲(浮点), 龙门升降脉冲当量(浮点）, 龙门升降当前位置(mm)

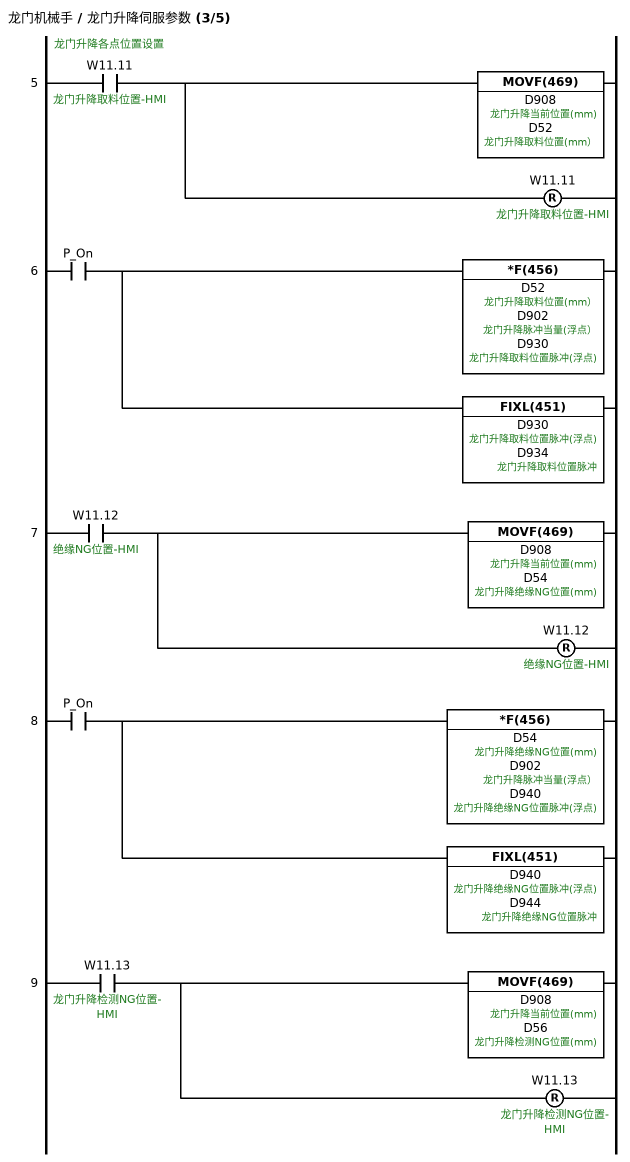
; rung 5: 龙门升降各点位置设置
LD W11.11  ; 龙门升降取料位置-HMI
MOVF(469) D908 D52  ; 龙门升降当前位置(mm), 龙门升降取料位置(mm）
RSET W11.11  ; 龙门升降取料位置-HMI
; rung 6
LD P_On
*F(456) D52 D902 D930  ; 龙门升降取料位置(mm）, 龙门升降脉冲当量(浮点）, 龙门升降取料位置脉冲(浮点)
FIXL(451) D930 D934  ; 龙门升降取料位置脉冲(浮点), 龙门升降取料位置脉冲
; rung 7
LD W11.12  ; 绝缘NG位置-HMI
MOVF(469) D908 D54  ; 龙门升降当前位置(mm), 龙门升降绝缘NG位置(mm)
RSET W11.12  ; 绝缘NG位置-HMI
; rung 8
LD P_On
*F(456) D54 D902 D940  ; 龙门升降绝缘NG位置(mm), 龙门升降脉冲当量(浮点）, 龙门升降绝缘NG位置脉冲(浮点)
FIXL(451) D940 D944  ; 龙门升降绝缘NG位置脉冲(浮点), 龙门升降绝缘NG位置脉冲
; rung 9
LD W11.13  ; 龙门升降检测NG位置-HMI
MOVF(469) D908 D56  ; 龙门升降当前位置(mm), 龙门升降检测NG位置(mm)
RSET W11.13  ; 龙门升降检测NG位置-HMI

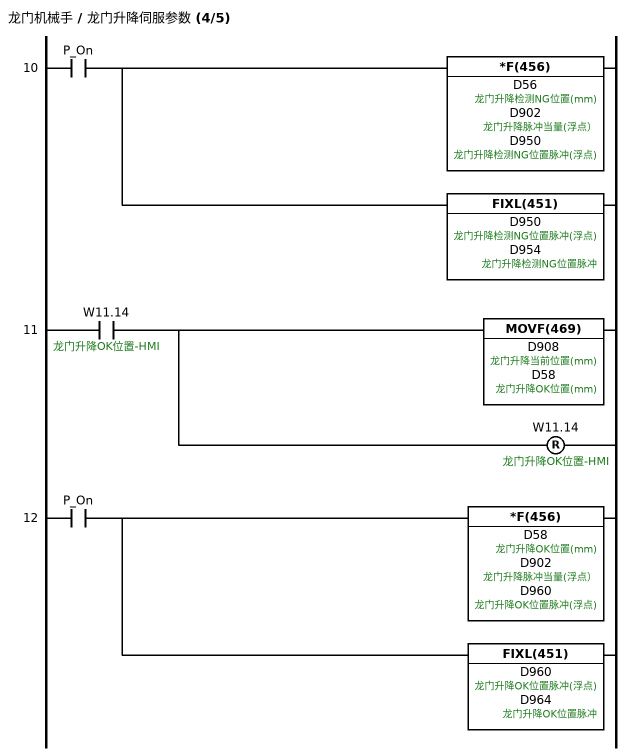
; rung 10
LD P_On
*F(456) D56 D902 D950  ; 龙门升降检测NG位置(mm), 龙门升降脉冲当量(浮点）, 龙门升降检测NG位置脉冲(浮点)
FIXL(451) D950 D954  ; 龙门升降检测NG位置脉冲(浮点), 龙门升降检测NG位置脉冲
; rung 11
LD W11.14  ; 龙门升降OK位置-HMI
MOVF(469) D908 D58  ; 龙门升降当前位置(mm), 龙门升降OK位置(mm)
RSET W11.14  ; 龙门升降OK位置-HMI
; rung 12
LD P_On
*F(456) D58 D902 D960  ; 龙门升降OK位置(mm), 龙门升降脉冲当量(浮点）, 龙门升降OK位置脉冲(浮点)
FIXL(451) D960 D964  ; 龙门升降OK位置脉冲(浮点), 龙门升降OK位置脉冲

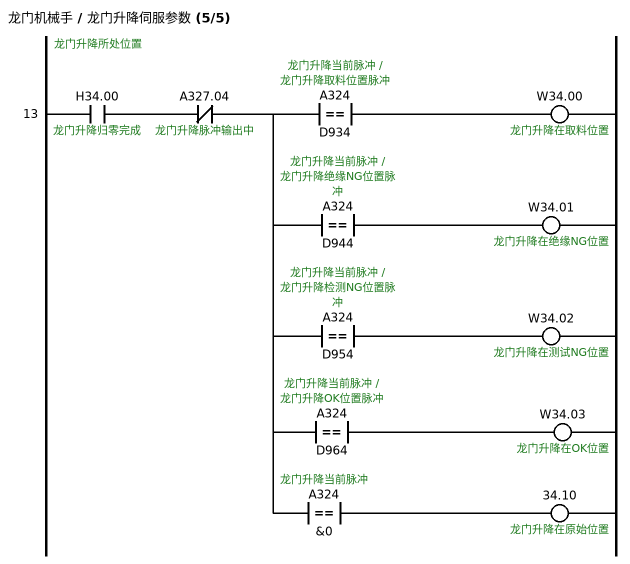
; rung 13: 龙门升降所处位置
LD H34.00  ; 龙门升降归零完成
ANDNOT A327.04  ; 龙门升降脉冲输出中
OUT TR0
AND=SL(303) A324 D934  ; 龙门升降当前脉冲, 龙门升降取料位置脉冲
OUT W34.00  ; 龙门升降在取料位置
LD TR0
AND=SL(303) A324 D944  ; 龙门升降当前脉冲, 龙门升降绝缘NG位置脉冲
OUT W34.01  ; 龙门升降在绝缘NG位置
LD TR0
AND=SL(303) A324 D954  ; 龙门升降当前脉冲, 龙门升降检测NG位置脉冲
OUT W34.02  ; 龙门升降在测试NG位置
LD TR0
AND=SL(303) A324 D964  ; 龙门升降当前脉冲, 龙门升降OK位置脉冲
OUT W34.03  ; 龙门升降在OK位置
LD TR0
AND=SL(303) A324 &0  ; 龙门升降当前脉冲
OUT 34.10  ; 龙门升降在原始位置

### Section 龙门前后伺服参数

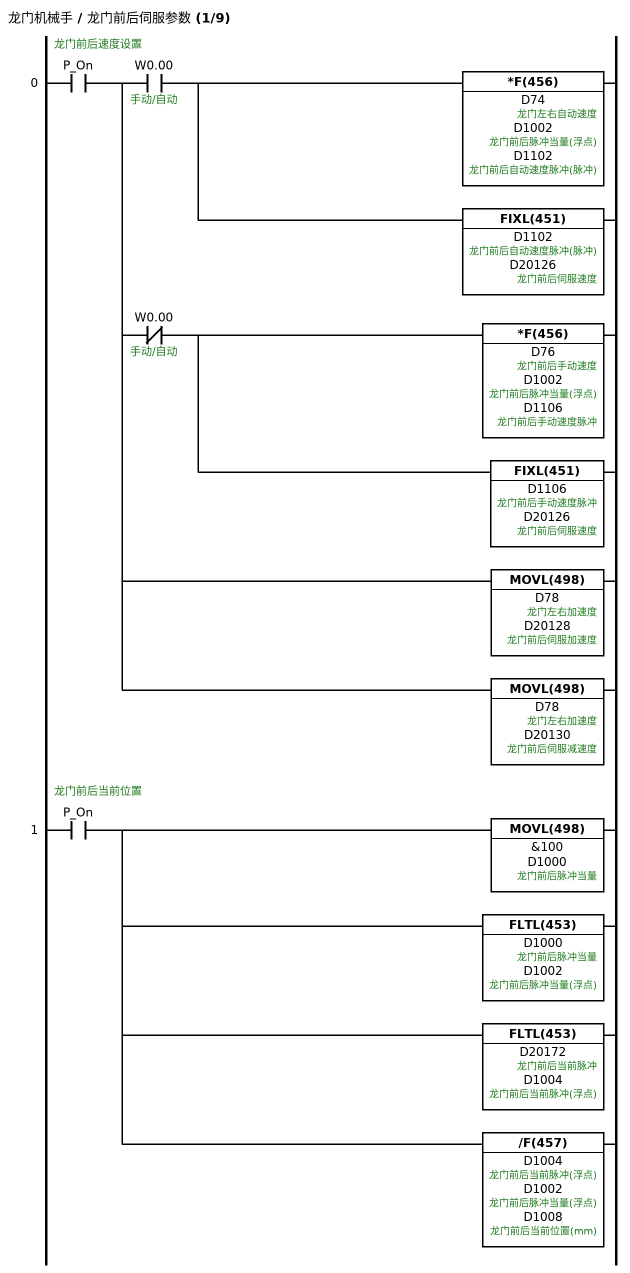
; rung 0: 龙门前后速度设置
LD P_On
OUT TR0
AND W0.00  ; 手动/自动
*F(456) D74 D1002 D1102  ; 龙门左右自动速度, 龙门前后脉冲当量(浮点), 龙门前后自动速度脉冲(脉冲)
FIXL(451) D1102 D20126  ; 龙门前后自动速度脉冲(脉冲), 龙门前后伺服速度
LD TR0
ANDNOT W0.00  ; 手动/自动
*F(456) D76 D1002 D1106  ; 龙门前后手动速度, 龙门前后脉冲当量(浮点), 龙门前后手动速度脉冲
FIXL(451) D1106 D20126  ; 龙门前后手动速度脉冲, 龙门前后伺服速度
LD TR0
MOVL(498) D78 D20128  ; 龙门左右加速度, 龙门前后伺服加速度
MOVL(498) D78 D20130  ; 龙门左右加速度, 龙门前后伺服减速度
; rung 1: 龙门前后当前位置
LD P_On
MOVL(498) &100 D1000  ; 龙门前后脉冲当量
FLTL(453) D1000 D1002  ; 龙门前后脉冲当量, 龙门前后脉冲当量(浮点)
FLTL(453) D20172 D1004  ; 龙门前后当前脉冲, 龙门前后当前脉冲(浮点)
/F(457) D1004 D1002 D1008  ; 龙门前后当前脉冲(浮点), 龙门前后脉冲当量(浮点), 龙门前后当前位置(mm)

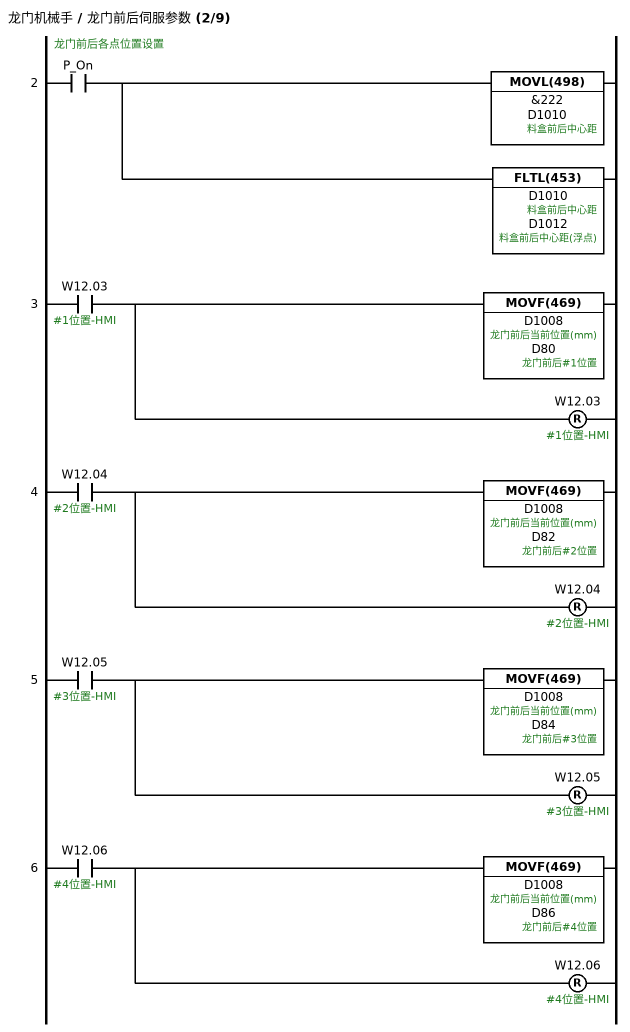
; rung 2: 龙门前后各点位置设置
LD P_On
MOVL(498) &222 D1010  ; 料盒前后中心距
FLTL(453) D1010 D1012  ; 料盒前后中心距, 料盒前后中心距(浮点)
; rung 3
LD W12.03  ; #1位置-HMI
MOVF(469) D1008 D80  ; 龙门前后当前位置(mm), 龙门前后#1位置
RSET W12.03  ; #1位置-HMI
; rung 4
LD W12.04  ; #2位置-HMI
MOVF(469) D1008 D82  ; 龙门前后当前位置(mm), 龙门前后#2位置
RSET W12.04  ; #2位置-HMI
; rung 5
LD W12.05  ; #3位置-HMI
MOVF(469) D1008 D84  ; 龙门前后当前位置(mm), 龙门前后#3位置
RSET W12.05  ; #3位置-HMI
; rung 6
LD W12.06  ; #4位置-HMI
MOVF(469) D1008 D86  ; 龙门前后当前位置(mm), 龙门前后#4位置
RSET W12.06  ; #4位置-HMI

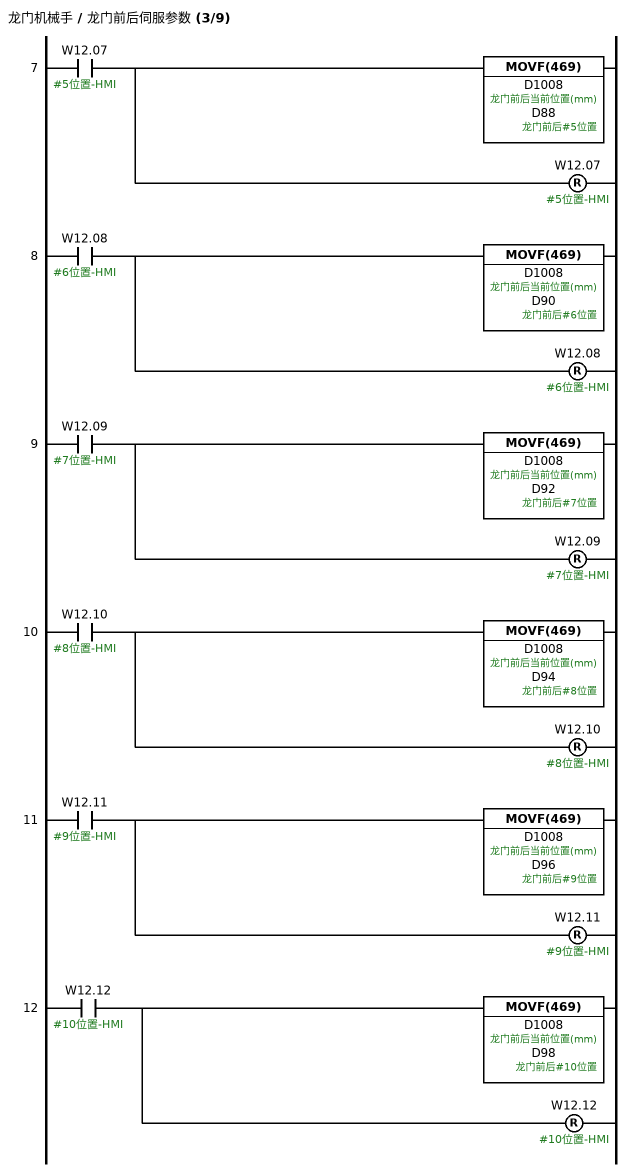
; rung 7
LD W12.07  ; #5位置-HMI
MOVF(469) D1008 D88  ; 龙门前后当前位置(mm), 龙门前后#5位置
RSET W12.07  ; #5位置-HMI
; rung 8
LD W12.08  ; #6位置-HMI
MOVF(469) D1008 D90  ; 龙门前后当前位置(mm), 龙门前后#6位置
RSET W12.08  ; #6位置-HMI
; rung 9
LD W12.09  ; #7位置-HMI
MOVF(469) D1008 D92  ; 龙门前后当前位置(mm), 龙门前后#7位置
RSET W12.09  ; #7位置-HMI
; rung 10
LD W12.10  ; #8位置-HMI
MOVF(469) D1008 D94  ; 龙门前后当前位置(mm), 龙门前后#8位置
RSET W12.10  ; #8位置-HMI
; rung 11
LD W12.11  ; #9位置-HMI
MOVF(469) D1008 D96  ; 龙门前后当前位置(mm), 龙门前后#9位置
RSET W12.11  ; #9位置-HMI
; rung 12
LD W12.12  ; #10位置-HMI
MOVF(469) D1008 D98  ; 龙门前后当前位置(mm), 龙门前后#10位置
RSET W12.12  ; #10位置-HMI

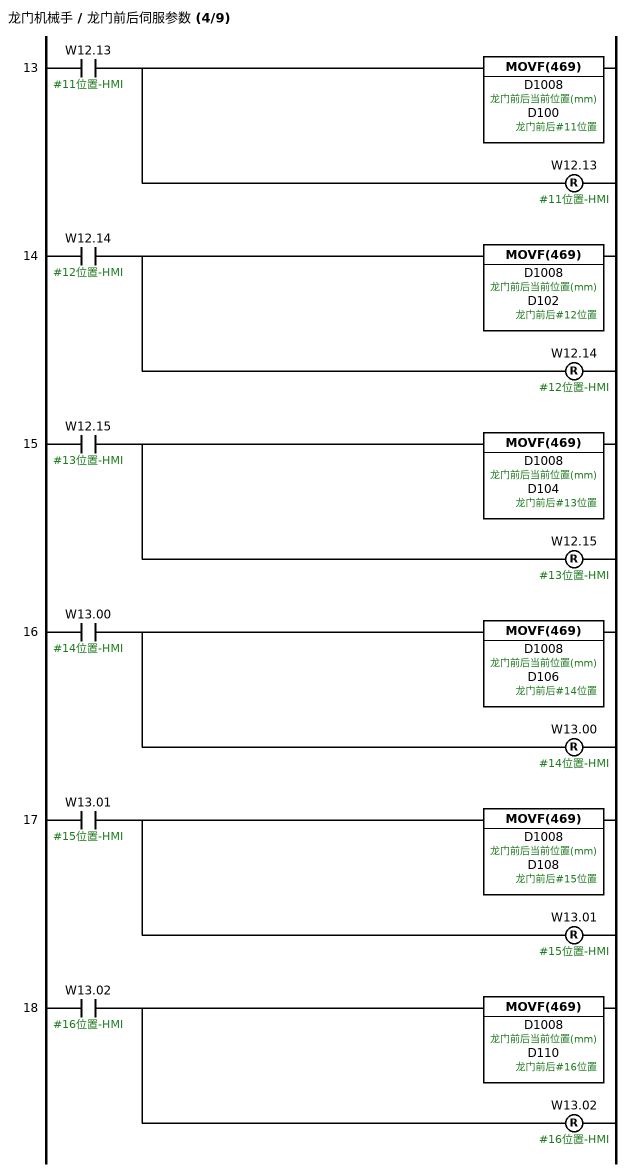
; rung 13
LD W12.13  ; #11位置-HMI
MOVF(469) D1008 D100  ; 龙门前后当前位置(mm), 龙门前后#11位置
RSET W12.13  ; #11位置-HMI
; rung 14
LD W12.14  ; #12位置-HMI
MOVF(469) D1008 D102  ; 龙门前后当前位置(mm), 龙门前后#12位置
RSET W12.14  ; #12位置-HMI
; rung 15
LD W12.15  ; #13位置-HMI
MOVF(469) D1008 D104  ; 龙门前后当前位置(mm), 龙门前后#13位置
RSET W12.15  ; #13位置-HMI
; rung 16
LD W13.00  ; #14位置-HMI
MOVF(469) D1008 D106  ; 龙门前后当前位置(mm), 龙门前后#14位置
RSET W13.00  ; #14位置-HMI
; rung 17
LD W13.01  ; #15位置-HMI
MOVF(469) D1008 D108  ; 龙门前后当前位置(mm), 龙门前后#15位置
RSET W13.01  ; #15位置-HMI
; rung 18
LD W13.02  ; #16位置-HMI
MOVF(469) D1008 D110  ; 龙门前后当前位置(mm), 龙门前后#16位置
RSET W13.02  ; #16位置-HMI

